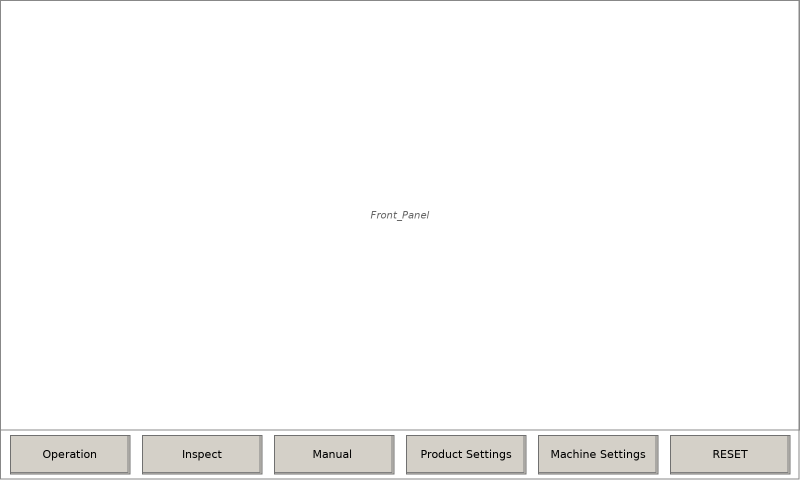
VISUALIZATION Visualization  // 800x480
    Button (10,435 120x39), "Operation"
        OnMouseClick: FrameSelectionChange Selection=SelectedFrame=9a7dff5b-3db9-4aa8-8ed3-29e44fa354e5, GlobSel=AssignType=Directly, SelType=Locally
        OnMouseClick: execute {
            MAIN.eModeCommand := E_PMLProtectedUnitMode.ePMLProtUnitMode_Production;
            MAIN.bOperation := TRUE;
            MAIN.bInspect := FALSE;
        }
    Button (274,435 120x39), "Manual"
        OnMouseClick: FrameSelectionChange Selection=SelectedFrame=9a7dff5b-3db9-4aa8-8ed3-29e44fa354e5, Selection=1, GlobSel=AssignType=Directly, SelType=Locally
        OnMouseClick: execute { Main.eModeCommand := E_PMLProtectedUnitMode.ePMLProtUnitMode_Manual; Main.bManual := TRUE; }
    Button (538,435 120x39), "Machine Settings"
        OnMouseClick: FrameSelectionChange Selection=SelectedFrame=9a7dff5b-3db9-4aa8-8ed3-29e44fa354e5, Selection=3, GlobSel=AssignType=Directly, SelType=Locally
        OnMouseClick: execute { MAIN.bMachineSettings := TRUE; }
    Frame (0,0 800x430)
        shows Front_Panel()
        shows ManualControl()
        shows Settings()
        shows MachineSettings()
        shows Manual_Inspect()
    Button (670,435 120x39), "RESET"
        OnMouseClick: execute { MAIN.hmiReset := TRUE; }
    Button (406,435 120x39), "Product Settings"
        OnMouseClick: FrameSelectionChange Selection=SelectedFrame=9a7dff5b-3db9-4aa8-8ed3-29e44fa354e5, Selection=2, GlobSel=AssignType=Directly, SelType=Locally
        OnMouseClick: execute { MAIN.bProductSettings := TRUE; }
    Button (142,435 120x39), "Inspect"
        OnMouseClick: FrameSelectionChange Selection=SelectedFrame=9a7dff5b-3db9-4aa8-8ed3-29e44fa354e5, Selection=4, GlobSel=AssignType=Directly, SelType=Locally
        OnMouseClick: execute {
            MAIN.eModeCommand := E_PMLProtectedUnitMode.ePMLProtUnitMode_Production;
            MAIN.bOperation := TRUE;
            MAIN.bInspect := TRUE;
        }
END_VISUALIZATION

(* stored: Version 1.1.0.1, ProductVersion 3.1.4024.5
   Visu Visualization: Id {b3142508-9b3b-48cc-a79a-eac45c569f44} *)
